// TIA Portal V16 export
// export: Created 2020-03-18T17:51:55.5456973Z, ExportSetting None, DisplayName Totally Integrated Automation Portal, DisplayVersion V16, DisplayName TIA Portal Version Control Interface, DisplayVersion V16, DisplayName TIA Portal Openness, DisplayVersion V16, DisplayName STEP 7 Professional, DisplayVersion V16, DisplayName STEP 7 Safety, DisplayVersion V16, DisplayName WinCC Advanced, DisplayVersion V16
DATA_BLOCK "DB_R134a_1_StepData"   // DB1310
{ S7_Optimized_Access := 'TRUE' }
AUTHOR : JMP/CSS
VERSION : 7.1
// stored: AutoNumber false, MemoryReserve 100
   VAR RETAIN
      Timestamp : Date_And_Time := DT#2019-07-18-09:28:16;
      DescriptionMedium : Array[1..4] of WString[36];
      "Step" { S7_SetPoint := 'True'} : Array[0..68] of "UDT_STEP_DATA";
      Values { S7_SetPoint := 'True'} : "UDT_CYCLE_VALUES";
      Valve { S7_SetPoint := 'True'} : Array[1..64] of "UDT_VISU_VALVE_NAMES";
      ParaInfo { S7_SetPoint := 'True'} : Array[1..15] of "UDT_STEP_DATA_PARA_VISU";
   END_VAR
BEGIN
   DescriptionMedium[1..2] := WSTRING#'R134a';
   DescriptionMedium[3] := WSTRING#'空调r134a';
   DescriptionMedium[4] := WSTRING#'Übersetzung fehlt';
   "Step"[0].NextStep := 4;
   "Step"[1..3].NextStep := 0;
   "Step"[4].NextStep := 10;
   "Step"[5..9].NextStep := 0;
   "Step"[10].NextStep := 11;
   "Step"[11].NextStep := 15;
   "Step"[12..14].NextStep := 0;
   "Step"[15].NextStep := 16;
   "Step"[16].NextStep := 20;
   "Step"[17].NextStep := 62;
   "Step"[18..19].NextStep := 0;
   "Step"[20].NextStep := 21;
   "Step"[21].NextStep := 22;
   "Step"[22].NextStep := 27;
   "Step"[23..26].NextStep := 0;
   "Step"[27].NextStep := 28;
   "Step"[28].NextStep := 29;
   "Step"[29].NextStep := 30;
   "Step"[30].NextStep := 31;
   "Step"[31].NextStep := 32;
   "Step"[32].NextStep := 33;
   "Step"[33].NextStep := 34;
   "Step"[34].NextStep := 35;
   "Step"[35].NextStep := 36;
   "Step"[36].NextStep := 37;
   "Step"[37].NextStep := 38;
   "Step"[38].NextStep := 39;
   "Step"[39].NextStep := 62;
   "Step"[40..61].NextStep := 0;
   "Step"[62].NextStep := 64;
   "Step"[63].NextStep := 0;
   "Step"[64].NextStep := 66;
   "Step"[65..68].NextStep := 0;
   "Step"[0..9].AbortStep := 0;
   "Step"[10..11].AbortStep := 62;
   "Step"[12..14].AbortStep := 0;
   "Step"[15].AbortStep := 62;
   "Step"[16].AbortStep := 17;
   "Step"[17].AbortStep := 62;
   "Step"[18..19].AbortStep := 0;
   "Step"[20..22].AbortStep := 27;
   "Step"[23..26].AbortStep := 0;
   "Step"[27].AbortStep := 28;
   "Step"[28..29].AbortStep := 62;
   "Step"[30..37].AbortStep := 17;
   "Step"[38].AbortStep := 39;
   "Step"[39].AbortStep := 62;
   "Step"[40..61].AbortStep := 0;
   "Step"[62].AbortStep := 64;
   "Step"[63..68].AbortStep := 0;
   "Step"[0..9].OptionStep := 0;
   "Step"[10].OptionStep := 15;
   "Step"[11..15].OptionStep := 0;
   "Step"[16].OptionStep := 29;
   "Step"[17..34].OptionStep := 0;
   "Step"[35].OptionStep := 37;
   "Step"[36].OptionStep := 0;
   "Step"[37].OptionStep := 57;
   "Step"[38..68].OptionStep := 0;
   "Step"[0..9].WaitingTime := 0;
   "Step"[10..11].WaitingTime := 1000;
   "Step"[12..14].WaitingTime := 0;
   "Step"[15].WaitingTime := 1000;
   "Step"[16].WaitingTime := 3000;
   "Step"[17].WaitingTime := 5000;
   "Step"[18..19].WaitingTime := 0;
   "Step"[20].WaitingTime := 20000;
   "Step"[21].WaitingTime := 10000;
   "Step"[22].WaitingTime := 5000;
   "Step"[23..26].WaitingTime := 0;
   "Step"[27..28].WaitingTime := 5000;
   "Step"[29].WaitingTime := 4000;
   "Step"[30].WaitingTime := 10000;
   "Step"[31].WaitingTime := 15000;
   "Step"[32].WaitingTime := 1000;
   "Step"[33].WaitingTime := 4000;
   "Step"[34].WaitingTime := 5000;
   "Step"[35..36].WaitingTime := 1000;
   "Step"[37].WaitingTime := 0;
   "Step"[38].WaitingTime := 1000;
   "Step"[39].WaitingTime := 2000;
   "Step"[40..65].WaitingTime := 0;
   "Step"[66].WaitingTime := 5000;
   "Step"[67..68].WaitingTime := 0;
   "Step"[0..10].MonitoringTime := 0;
   "Step"[11].MonitoringTime := 4000;
   "Step"[12..15].MonitoringTime := 0;
   "Step"[16].MonitoringTime := 4000;
   "Step"[17..19].MonitoringTime := 0;
   "Step"[20].MonitoringTime := 23000;
   "Step"[21].MonitoringTime := 11000;
   "Step"[22].MonitoringTime := 6000;
   "Step"[23..26].MonitoringTime := 0;
   "Step"[27..28].MonitoringTime := 10000;
   "Step"[29].MonitoringTime := 5000;
   "Step"[30].MonitoringTime := 15000;
   "Step"[31].MonitoringTime := 45000;
   "Step"[32].MonitoringTime := 0;
   "Step"[33..34].MonitoringTime := 6000;
   "Step"[35].MonitoringTime := 0;
   "Step"[36].MonitoringTime := 20000;
   "Step"[37].MonitoringTime := 0;
   "Step"[38].MonitoringTime := 20000;
   "Step"[39..68].MonitoringTime := 0;
   "Step"[0].Setpoint[0..15] := 0;
   "Step"[1].Setpoint[0..15] := 0;
   "Step"[2].Setpoint[0..15] := 0;
   "Step"[3].Setpoint[0..15] := 0;
   "Step"[4].Setpoint[0..15] := 0;
   "Step"[5].Setpoint[0..15] := 0;
   "Step"[6].Setpoint[0..15] := 0;
   "Step"[7].Setpoint[0..15] := 0;
   "Step"[8].Setpoint[0..15] := 0;
   "Step"[9].Setpoint[0..15] := 0;
   "Step"[10].Setpoint[0..15] := 0;
   "Step"[11].Setpoint[0] := 0;
   "Step"[11].Setpoint[1] := 100;
   "Step"[11].Setpoint[2..15] := 0;
   "Step"[12].Setpoint[0..15] := 0;
   "Step"[13].Setpoint[0..15] := 0;
   "Step"[14].Setpoint[0..15] := 0;
   "Step"[15].Setpoint[0..15] := 0;
   "Step"[16].Setpoint[0..4] := 0;
   "Step"[16].Setpoint[5] := 1200;
   "Step"[16].Setpoint[6..15] := 0;
   "Step"[17].Setpoint[0..15] := 0;
   "Step"[18].Setpoint[0..15] := 0;
   "Step"[19].Setpoint[0..15] := 0;
   "Step"[20].Setpoint[0..4] := 0;
   "Step"[20].Setpoint[5] := 15000;
   "Step"[20].Setpoint[6..12] := 0;
   "Step"[20].Setpoint[13] := 15200;
   "Step"[20].Setpoint[14..15] := 0;
   "Step"[21].Setpoint[0..4] := 0;
   "Step"[21].Setpoint[5] := 15000;
   "Step"[21].Setpoint[6..12] := 0;
   "Step"[21].Setpoint[13] := 15200;
   "Step"[21].Setpoint[14..15] := 0;
   "Step"[22].Setpoint[0..4] := 0;
   "Step"[22].Setpoint[5] := 14900;
   "Step"[22].Setpoint[6] := -100;
   "Step"[22].Setpoint[7..12] := 0;
   "Step"[22].Setpoint[13] := 15200;
   "Step"[22].Setpoint[14..15] := 0;
   "Step"[23].Setpoint[0..15] := 0;
   "Step"[24].Setpoint[0..15] := 0;
   "Step"[25].Setpoint[0..15] := 0;
   "Step"[26].Setpoint[0..15] := 0;
   "Step"[27].Setpoint[0..4] := 0;
   "Step"[27].Setpoint[5] := 3000;
   "Step"[27].Setpoint[6..15] := 0;
   "Step"[28].Setpoint[0..4] := 0;
   "Step"[28].Setpoint[5] := 500;
   "Step"[28].Setpoint[6..15] := 0;
   "Step"[29].Setpoint[0] := 0;
   "Step"[29].Setpoint[1] := 10;
   "Step"[29].Setpoint[2..15] := 0;
   "Step"[30].Setpoint[0] := 0;
   "Step"[30].Setpoint[1] := 500;
   "Step"[30].Setpoint[2..15] := 0;
   "Step"[31].Setpoint[0] := 0;
   "Step"[31].Setpoint[1] := 30;
   "Step"[31].Setpoint[2..15] := 0;
   "Step"[32].Setpoint[0..15] := 0;
   "Step"[33].Setpoint[0] := 0;
   "Step"[33].Setpoint[1] := 50;
   "Step"[33].Setpoint[2] := 40;
   "Step"[33].Setpoint[3..15] := 0;
   "Step"[34].Setpoint[0] := 0;
   "Step"[34].Setpoint[1] := 50;
   "Step"[34].Setpoint[2..15] := 0;
   "Step"[35].Setpoint[0..15] := 0;
   "Step"[36].Setpoint[0..7] := 0;
   "Step"[36].Setpoint[8] := 15;
   "Step"[36].Setpoint[9..15] := 0;
   "Step"[37].Setpoint[0..15] := 0;
   "Step"[38].Setpoint[0..6] := 0;
   "Step"[38].Setpoint[7] := 550;
   "Step"[38].Setpoint[8..15] := 0;
   "Step"[39].Setpoint[0..15] := 0;
   "Step"[40].Setpoint[0..15] := 0;
   "Step"[41].Setpoint[0..15] := 0;
   "Step"[42].Setpoint[0..15] := 0;
   "Step"[43].Setpoint[0..15] := 0;
   "Step"[44].Setpoint[0..15] := 0;
   "Step"[45].Setpoint[0..15] := 0;
   "Step"[46].Setpoint[0..15] := 0;
   "Step"[47].Setpoint[0..15] := 0;
   "Step"[48].Setpoint[0..15] := 0;
   "Step"[49].Setpoint[0..15] := 0;
   "Step"[50].Setpoint[0..15] := 0;
   "Step"[51].Setpoint[0..15] := 0;
   "Step"[52].Setpoint[0..15] := 0;
   "Step"[53].Setpoint[0..15] := 0;
   "Step"[54].Setpoint[0..15] := 0;
   "Step"[55].Setpoint[0..15] := 0;
   "Step"[56].Setpoint[0..15] := 0;
   "Step"[57].Setpoint[0..15] := 0;
   "Step"[58].Setpoint[0..15] := 0;
   "Step"[59].Setpoint[0..15] := 0;
   "Step"[60].Setpoint[0..15] := 0;
   "Step"[61].Setpoint[0..15] := 0;
   "Step"[62].Setpoint[0..15] := 0;
   "Step"[63].Setpoint[0..15] := 0;
   "Step"[64].Setpoint[0..15] := 0;
   "Step"[65].Setpoint[0..15] := 0;
   "Step"[66].Setpoint[0..15] := 0;
   "Step"[67].Setpoint[0..15] := 0;
   "Step"[68].Setpoint[0..15] := 0;
   "Step"[0..9].History.ElapsedTime := 0;
   "Step"[10..11].History.ElapsedTime := 1001;
   "Step"[12..14].History.ElapsedTime := 0;
   "Step"[15].History.ElapsedTime := 1001;
   "Step"[16].History.ElapsedTime := 3001;
   "Step"[17..19].History.ElapsedTime := 0;
   "Step"[20].History.ElapsedTime := 20001;
   "Step"[21].History.ElapsedTime := 10001;
   "Step"[22].History.ElapsedTime := 5001;
   "Step"[23..26].History.ElapsedTime := 0;
   "Step"[27..28].History.ElapsedTime := 5001;
   "Step"[29].History.ElapsedTime := 4001;
   "Step"[30].History.ElapsedTime := 10001;
   "Step"[31].History.ElapsedTime := 15001;
   "Step"[32].History.ElapsedTime := 1001;
   "Step"[33].History.ElapsedTime := 4001;
   "Step"[34].History.ElapsedTime := 5001;
   "Step"[35].History.ElapsedTime := 1001;
   "Step"[36].History.ElapsedTime := 3545;
   "Step"[37].History.ElapsedTime := 1;
   "Step"[38..61].History.ElapsedTime := 0;
   "Step"[62].History.ElapsedTime := 65252;
   "Step"[63].History.ElapsedTime := 0;
   "Step"[64].History.ElapsedTime := 7412;
   "Step"[65].History.ElapsedTime := 0;
   "Step"[66].History.ElapsedTime := 5001;
   "Step"[67..68].History.ElapsedTime := 0;
   "Step"[0].History.Values[0] := 0;
   "Step"[0].History.Values[1] := 6;
   "Step"[0].History.Values[2] := 0;
   "Step"[0].History.Values[3] := 15522;
   "Step"[0].History.Values[4] := -1;
   "Step"[0].History.Values[5] := 54;
   "Step"[0].History.Values[6] := -1;
   "Step"[0].History.Values[7] := 0;
   "Step"[0].History.Values[8] := 15;
   "Step"[0].History.Values[9..15] := 0;
   "Step"[1].History.Values[0..15] := 0;
   "Step"[2].History.Values[0..15] := 0;
   "Step"[3].History.Values[0..15] := 0;
   "Step"[4].History.Values[0..15] := 0;
   "Step"[5].History.Values[0..15] := 0;
   "Step"[6].History.Values[0..15] := 0;
   "Step"[7].History.Values[0..15] := 0;
   "Step"[8].History.Values[0..15] := 0;
   "Step"[9].History.Values[0..15] := 0;
   "Step"[10].History.Values[0] := 0;
   "Step"[10].History.Values[1..2] := 7;
   "Step"[10].History.Values[3..4] := 15524;
   "Step"[10].History.Values[5..6] := -700;
   "Step"[10].History.Values[7..15] := 0;
   "Step"[11].History.Values[0] := 0;
   "Step"[11].History.Values[1] := 10;
   "Step"[11].History.Values[2] := 3;
   "Step"[11].History.Values[3] := 15524;
   "Step"[11].History.Values[4] := 0;
   "Step"[11].History.Values[5] := -700;
   "Step"[11].History.Values[6..15] := 0;
   "Step"[12].History.Values[0..15] := 0;
   "Step"[13].History.Values[0..15] := 0;
   "Step"[14].History.Values[0..15] := 0;
   "Step"[15].History.Values[0] := 0;
   "Step"[15].History.Values[1] := 7;
   "Step"[15].History.Values[2] := -3;
   "Step"[15].History.Values[3] := 15524;
   "Step"[15].History.Values[4] := 0;
   "Step"[15].History.Values[5] := -700;
   "Step"[15].History.Values[6..15] := 0;
   "Step"[16].History.Values[0] := 0;
   "Step"[16].History.Values[1] := 6;
   "Step"[16].History.Values[2] := -1;
   "Step"[16].History.Values[3] := 15524;
   "Step"[16].History.Values[4] := 0;
   "Step"[16].History.Values[5] := -40;
   "Step"[16].History.Values[6] := 660;
   "Step"[16].History.Values[7..15] := 0;
   "Step"[17].History.Values[0..15] := 0;
   "Step"[18].History.Values[0..15] := 0;
   "Step"[19].History.Values[0..15] := 0;
   "Step"[20].History.Values[0] := 0;
   "Step"[20].History.Values[1] := 6;
   "Step"[20].History.Values[2] := 0;
   "Step"[20].History.Values[3] := 15524;
   "Step"[20].History.Values[4] := 0;
   "Step"[20].History.Values[5] := 15231;
   "Step"[20].History.Values[6] := 15271;
   "Step"[20].History.Values[7..12] := 0;
   "Step"[20].History.Values[13] := 15200;
   "Step"[20].History.Values[14..15] := 0;
   "Step"[21].History.Values[0] := 0;
   "Step"[21].History.Values[1] := 6;
   "Step"[21].History.Values[2] := 0;
   "Step"[21].History.Values[3] := 15523;
   "Step"[21].History.Values[4] := -1;
   "Step"[21].History.Values[5] := 15230;
   "Step"[21].History.Values[6] := -1;
   "Step"[21].History.Values[7..12] := 0;
   "Step"[21].History.Values[13] := 15200;
   "Step"[21].History.Values[14..15] := 0;
   "Step"[22].History.Values[0] := 0;
   "Step"[22].History.Values[1] := 6;
   "Step"[22].History.Values[2] := 0;
   "Step"[22].History.Values[3] := 15524;
   "Step"[22].History.Values[4] := 1;
   "Step"[22].History.Values[5] := 15231;
   "Step"[22].History.Values[6] := 1;
   "Step"[22].History.Values[7..12] := 0;
   "Step"[22].History.Values[13] := 15200;
   "Step"[22].History.Values[14..15] := 0;
   "Step"[23].History.Values[0..15] := 0;
   "Step"[24].History.Values[0..15] := 0;
   "Step"[25].History.Values[0..15] := 0;
   "Step"[26].History.Values[0..15] := 0;
   "Step"[27].History.Values[0] := 0;
   "Step"[27].History.Values[1] := 6;
   "Step"[27].History.Values[2] := 0;
   "Step"[27].History.Values[3] := 15523;
   "Step"[27].History.Values[4] := -1;
   "Step"[27].History.Values[5] := 46;
   "Step"[27].History.Values[6] := -15185;
   "Step"[27].History.Values[7..15] := 0;
   "Step"[28].History.Values[0] := 0;
   "Step"[28].History.Values[1] := 6;
   "Step"[28].History.Values[2] := 0;
   "Step"[28].History.Values[3] := 15523;
   "Step"[28].History.Values[4] := 0;
   "Step"[28].History.Values[5] := 47;
   "Step"[28].History.Values[6] := 1;
   "Step"[28].History.Values[7..15] := 0;
   "Step"[29].History.Values[0] := 0;
   "Step"[29].History.Values[1] := 19;
   "Step"[29].History.Values[2] := 13;
   "Step"[29].History.Values[3] := 15523;
   "Step"[29].History.Values[4] := 0;
   "Step"[29].History.Values[5] := -722;
   "Step"[29].History.Values[6] := -769;
   "Step"[29].History.Values[7..15] := 0;
   "Step"[30].History.Values[0] := 0;
   "Step"[30].History.Values[1] := 13;
   "Step"[30].History.Values[2] := -6;
   "Step"[30].History.Values[3] := 15523;
   "Step"[30].History.Values[4] := 0;
   "Step"[30].History.Values[5] := -716;
   "Step"[30].History.Values[6] := 6;
   "Step"[30].History.Values[7..15] := 0;
   "Step"[31].History.Values[0] := 0;
   "Step"[31].History.Values[1] := 10;
   "Step"[31].History.Values[2] := -3;
   "Step"[31].History.Values[3] := 15523;
   "Step"[31].History.Values[4] := 0;
   "Step"[31].History.Values[5] := -712;
   "Step"[31].History.Values[6] := 4;
   "Step"[31].History.Values[7..15] := 0;
   "Step"[32].History.Values[0] := 0;
   "Step"[32].History.Values[1] := 14;
   "Step"[32].History.Values[2] := 4;
   "Step"[32].History.Values[3] := 15523;
   "Step"[32].History.Values[4] := 0;
   "Step"[32].History.Values[5] := -711;
   "Step"[32].History.Values[6] := 1;
   "Step"[32].History.Values[7..15] := 0;
   "Step"[33].History.Values[0] := 0;
   "Step"[33].History.Values[1] := 22;
   "Step"[33].History.Values[2] := 8;
   "Step"[33].History.Values[3] := 15523;
   "Step"[33].History.Values[4] := 0;
   "Step"[33].History.Values[5] := -710;
   "Step"[33].History.Values[6] := 1;
   "Step"[33].History.Values[7..15] := 0;
   "Step"[34].History.Values[0] := 0;
   "Step"[34].History.Values[1] := 10;
   "Step"[34].History.Values[2] := -12;
   "Step"[34].History.Values[3] := 15523;
   "Step"[34].History.Values[4] := 0;
   "Step"[34].History.Values[5] := -710;
   "Step"[34].History.Values[6..15] := 0;
   "Step"[35].History.Values[0] := 0;
   "Step"[35].History.Values[1] := 7;
   "Step"[35].History.Values[2] := -3;
   "Step"[35].History.Values[3] := 15523;
   "Step"[35].History.Values[4] := 0;
   "Step"[35].History.Values[5] := -709;
   "Step"[35].History.Values[6] := 1;
   "Step"[35].History.Values[7..15] := 0;
   "Step"[36].History.Values[0] := 0;
   "Step"[36].History.Values[1] := 6;
   "Step"[36].History.Values[2] := -1;
   "Step"[36].History.Values[3] := 15523;
   "Step"[36].History.Values[4] := 0;
   "Step"[36].History.Values[5] := -708;
   "Step"[36].History.Values[6] := 1;
   "Step"[36].History.Values[7] := 0;
   "Step"[36].History.Values[8] := 14;
   "Step"[36].History.Values[9..15] := 0;
   "Step"[37].History.Values[0] := 0;
   "Step"[37].History.Values[1] := 6;
   "Step"[37].History.Values[2] := 0;
   "Step"[37].History.Values[3] := 15523;
   "Step"[37].History.Values[4] := 0;
   "Step"[37].History.Values[5] := -708;
   "Step"[37].History.Values[6..7] := 0;
   "Step"[37].History.Values[8] := 15;
   "Step"[37].History.Values[9..15] := 0;
   "Step"[38].History.Values[0..15] := 0;
   "Step"[39].History.Values[0..15] := 0;
   "Step"[40].History.Values[0..15] := 0;
   "Step"[41].History.Values[0..15] := 0;
   "Step"[42].History.Values[0..15] := 0;
   "Step"[43].History.Values[0..15] := 0;
   "Step"[44].History.Values[0..15] := 0;
   "Step"[45].History.Values[0..15] := 0;
   "Step"[46].History.Values[0..15] := 0;
   "Step"[47].History.Values[0..15] := 0;
   "Step"[48].History.Values[0..15] := 0;
   "Step"[49].History.Values[0..15] := 0;
   "Step"[50].History.Values[0..15] := 0;
   "Step"[51].History.Values[0..15] := 0;
   "Step"[52].History.Values[0..15] := 0;
   "Step"[53].History.Values[0..15] := 0;
   "Step"[54].History.Values[0..15] := 0;
   "Step"[55].History.Values[0..15] := 0;
   "Step"[56].History.Values[0..15] := 0;
   "Step"[57].History.Values[0..15] := 0;
   "Step"[58].History.Values[0..15] := 0;
   "Step"[59].History.Values[0..15] := 0;
   "Step"[60].History.Values[0..15] := 0;
   "Step"[61].History.Values[0..15] := 0;
   "Step"[62].History.Values[0] := 0;
   "Step"[62].History.Values[1] := 6;
   "Step"[62].History.Values[2] := 0;
   "Step"[62].History.Values[3] := 15523;
   "Step"[62].History.Values[4] := 0;
   "Step"[62].History.Values[5] := -698;
   "Step"[62].History.Values[6] := 10;
   "Step"[62].History.Values[7] := 0;
   "Step"[62].History.Values[8] := 15;
   "Step"[62].History.Values[9..15] := 0;
   "Step"[63].History.Values[0..15] := 0;
   "Step"[64].History.Values[0] := 0;
   "Step"[64].History.Values[1] := 6;
   "Step"[64].History.Values[2] := 0;
   "Step"[64].History.Values[3] := 15523;
   "Step"[64].History.Values[4] := 0;
   "Step"[64].History.Values[5] := 55;
   "Step"[64].History.Values[6] := 753;
   "Step"[64].History.Values[7] := 0;
   "Step"[64].History.Values[8] := 15;
   "Step"[64].History.Values[9..15] := 0;
   "Step"[65].History.Values[0..15] := 0;
   "Step"[66].History.Values[0] := 0;
   "Step"[66].History.Values[1] := 6;
   "Step"[66].History.Values[2] := 0;
   "Step"[66].History.Values[3] := 15522;
   "Step"[66].History.Values[4] := -1;
   "Step"[66].History.Values[5] := 54;
   "Step"[66].History.Values[6] := -1;
   "Step"[66].History.Values[7] := 0;
   "Step"[66].History.Values[8] := 15;
   "Step"[66].History.Values[9..15] := 0;
   "Step"[67].History.Values[0..15] := 0;
   "Step"[68].History.Values[0..15] := 0;
   "Step"[0].Valve[0..9] := FALSE;
   "Step"[0].Valve[10] := TRUE;
   "Step"[0].Valve[11] := FALSE;
   "Step"[0].Valve[12] := TRUE;
   "Step"[0].Valve[13..15] := FALSE;
   "Step"[0].Valve[16..21] := TRUE;
   "Step"[0].Valve[22] := FALSE;
   "Step"[0].Valve[23..24] := TRUE;
   "Step"[0].Valve[25..42] := FALSE;
   "Step"[0].Valve[43..45] := TRUE;
   "Step"[0].Valve[46..64] := FALSE;
   "Step"[1].Valve[0..64] := FALSE;
   "Step"[2].Valve[0..64] := FALSE;
   "Step"[3].Valve[0..64] := FALSE;
   "Step"[4].Valve[0..9] := FALSE;
   "Step"[4].Valve[10] := TRUE;
   "Step"[4].Valve[11] := FALSE;
   "Step"[4].Valve[12] := TRUE;
   "Step"[4].Valve[13..15] := FALSE;
   "Step"[4].Valve[16..21] := TRUE;
   "Step"[4].Valve[22] := FALSE;
   "Step"[4].Valve[23..24] := TRUE;
   "Step"[4].Valve[25..42] := FALSE;
   "Step"[4].Valve[43..46] := TRUE;
   "Step"[4].Valve[47..52] := FALSE;
   "Step"[4].Valve[53] := TRUE;
   "Step"[4].Valve[54..59] := FALSE;
   "Step"[4].Valve[60] := TRUE;
   "Step"[4].Valve[61..64] := FALSE;
   "Step"[5].Valve[0..64] := FALSE;
   "Step"[6].Valve[0..64] := FALSE;
   "Step"[7].Valve[0..64] := FALSE;
   "Step"[8].Valve[0..64] := FALSE;
   "Step"[9].Valve[0..64] := FALSE;
   "Step"[10].Valve[0..9] := FALSE;
   "Step"[10].Valve[10] := TRUE;
   "Step"[10].Valve[11] := FALSE;
   "Step"[10].Valve[12] := TRUE;
   "Step"[10].Valve[13..15] := FALSE;
   "Step"[10].Valve[16..21] := TRUE;
   "Step"[10].Valve[22] := FALSE;
   "Step"[10].Valve[23..24] := TRUE;
   "Step"[10].Valve[25..42] := FALSE;
   "Step"[10].Valve[43..45] := TRUE;
   "Step"[10].Valve[46..56] := FALSE;
   "Step"[10].Valve[57] := TRUE;
   "Step"[10].Valve[58..61] := FALSE;
   "Step"[10].Valve[62] := TRUE;
   "Step"[10].Valve[63..64] := FALSE;
   "Step"[11].Valve[0..9] := FALSE;
   "Step"[11].Valve[10] := TRUE;
   "Step"[11].Valve[11] := FALSE;
   "Step"[11].Valve[12] := TRUE;
   "Step"[11].Valve[13..15] := FALSE;
   "Step"[11].Valve[16..21] := TRUE;
   "Step"[11].Valve[22] := FALSE;
   "Step"[11].Valve[23..24] := TRUE;
   "Step"[11].Valve[25..42] := FALSE;
   "Step"[11].Valve[43..46] := TRUE;
   "Step"[11].Valve[47..52] := FALSE;
   "Step"[11].Valve[53] := TRUE;
   "Step"[11].Valve[54..56] := FALSE;
   "Step"[11].Valve[57] := TRUE;
   "Step"[11].Valve[58..59] := FALSE;
   "Step"[11].Valve[60] := TRUE;
   "Step"[11].Valve[61] := FALSE;
   "Step"[11].Valve[62] := TRUE;
   "Step"[11].Valve[63..64] := FALSE;
   "Step"[12].Valve[0..64] := FALSE;
   "Step"[13].Valve[0..64] := FALSE;
   "Step"[14].Valve[0..64] := FALSE;
   "Step"[15].Valve[0..9] := FALSE;
   "Step"[15].Valve[10] := TRUE;
   "Step"[15].Valve[11] := FALSE;
   "Step"[15].Valve[12] := TRUE;
   "Step"[15].Valve[13..15] := FALSE;
   "Step"[15].Valve[16..21] := TRUE;
   "Step"[15].Valve[22] := FALSE;
   "Step"[15].Valve[23..24] := TRUE;
   "Step"[15].Valve[25..42] := FALSE;
   "Step"[15].Valve[43..45] := TRUE;
   "Step"[15].Valve[46..52] := FALSE;
   "Step"[15].Valve[53] := TRUE;
   "Step"[15].Valve[54..56] := FALSE;
   "Step"[15].Valve[57] := TRUE;
   "Step"[15].Valve[58..59] := FALSE;
   "Step"[15].Valve[60] := TRUE;
   "Step"[15].Valve[61] := FALSE;
   "Step"[15].Valve[62] := TRUE;
   "Step"[15].Valve[63..64] := FALSE;
   "Step"[16].Valve[0..9] := FALSE;
   "Step"[16].Valve[10] := TRUE;
   "Step"[16].Valve[11] := FALSE;
   "Step"[16].Valve[12] := TRUE;
   "Step"[16].Valve[13..15] := FALSE;
   "Step"[16].Valve[16..21] := TRUE;
   "Step"[16].Valve[22] := FALSE;
   "Step"[16].Valve[23..24] := TRUE;
   "Step"[16].Valve[25..42] := FALSE;
   "Step"[16].Valve[43..45] := TRUE;
   "Step"[16].Valve[46..52] := FALSE;
   "Step"[16].Valve[53] := TRUE;
   "Step"[16].Valve[54..55] := FALSE;
   "Step"[16].Valve[56..57] := TRUE;
   "Step"[16].Valve[58..59] := FALSE;
   "Step"[16].Valve[60..62] := TRUE;
   "Step"[16].Valve[63..64] := FALSE;
   "Step"[17].Valve[0..9] := FALSE;
   "Step"[17].Valve[10] := TRUE;
   "Step"[17].Valve[11] := FALSE;
   "Step"[17].Valve[12] := TRUE;
   "Step"[17].Valve[13..15] := FALSE;
   "Step"[17].Valve[16..21] := TRUE;
   "Step"[17].Valve[22] := FALSE;
   "Step"[17].Valve[23..24] := TRUE;
   "Step"[17].Valve[25..42] := FALSE;
   "Step"[17].Valve[43..45] := TRUE;
   "Step"[17].Valve[46..48] := FALSE;
   "Step"[17].Valve[49] := TRUE;
   "Step"[17].Valve[50..52] := FALSE;
   "Step"[17].Valve[53] := TRUE;
   "Step"[17].Valve[54..56] := FALSE;
   "Step"[17].Valve[57] := TRUE;
   "Step"[17].Valve[58..59] := FALSE;
   "Step"[17].Valve[60] := TRUE;
   "Step"[17].Valve[61] := FALSE;
   "Step"[17].Valve[62] := TRUE;
   "Step"[17].Valve[63..64] := FALSE;
   "Step"[18].Valve[0..64] := FALSE;
   "Step"[19].Valve[0..64] := FALSE;
   "Step"[20].Valve[0..9] := FALSE;
   "Step"[20].Valve[10] := TRUE;
   "Step"[20].Valve[11] := FALSE;
   "Step"[20].Valve[12] := TRUE;
   "Step"[20].Valve[13..15] := FALSE;
   "Step"[20].Valve[16..21] := TRUE;
   "Step"[20].Valve[22] := FALSE;
   "Step"[20].Valve[23..24] := TRUE;
   "Step"[20].Valve[25..42] := FALSE;
   "Step"[20].Valve[43..45] := TRUE;
   "Step"[20].Valve[46] := FALSE;
   "Step"[20].Valve[47] := TRUE;
   "Step"[20].Valve[48..52] := FALSE;
   "Step"[20].Valve[53] := TRUE;
   "Step"[20].Valve[54..55] := FALSE;
   "Step"[20].Valve[56..57] := TRUE;
   "Step"[20].Valve[58..59] := FALSE;
   "Step"[20].Valve[60..62] := TRUE;
   "Step"[20].Valve[63..64] := FALSE;
   "Step"[21].Valve[0..9] := FALSE;
   "Step"[21].Valve[10] := TRUE;
   "Step"[21].Valve[11] := FALSE;
   "Step"[21].Valve[12] := TRUE;
   "Step"[21].Valve[13..15] := FALSE;
   "Step"[21].Valve[16..21] := TRUE;
   "Step"[21].Valve[22] := FALSE;
   "Step"[21].Valve[23..24] := TRUE;
   "Step"[21].Valve[25..42] := FALSE;
   "Step"[21].Valve[43..45] := TRUE;
   "Step"[21].Valve[46] := FALSE;
   "Step"[21].Valve[47] := TRUE;
   "Step"[21].Valve[48..52] := FALSE;
   "Step"[21].Valve[53] := TRUE;
   "Step"[21].Valve[54..55] := FALSE;
   "Step"[21].Valve[56..57] := TRUE;
   "Step"[21].Valve[58..59] := FALSE;
   "Step"[21].Valve[60..62] := TRUE;
   "Step"[21].Valve[63..64] := FALSE;
   "Step"[22].Valve[0..9] := FALSE;
   "Step"[22].Valve[10] := TRUE;
   "Step"[22].Valve[11] := FALSE;
   "Step"[22].Valve[12] := TRUE;
   "Step"[22].Valve[13..15] := FALSE;
   "Step"[22].Valve[16..21] := TRUE;
   "Step"[22].Valve[22] := FALSE;
   "Step"[22].Valve[23..24] := TRUE;
   "Step"[22].Valve[25..42] := FALSE;
   "Step"[22].Valve[43..45] := TRUE;
   "Step"[22].Valve[46..52] := FALSE;
   "Step"[22].Valve[53] := TRUE;
   "Step"[22].Valve[54..55] := FALSE;
   "Step"[22].Valve[56..57] := TRUE;
   "Step"[22].Valve[58..59] := FALSE;
   "Step"[22].Valve[60..62] := TRUE;
   "Step"[22].Valve[63..64] := FALSE;
   "Step"[23].Valve[0..64] := FALSE;
   "Step"[24].Valve[0..64] := FALSE;
   "Step"[25].Valve[0..64] := FALSE;
   "Step"[26].Valve[0..64] := FALSE;
   "Step"[27].Valve[0..9] := FALSE;
   "Step"[27].Valve[10] := TRUE;
   "Step"[27].Valve[11] := FALSE;
   "Step"[27].Valve[12] := TRUE;
   "Step"[27].Valve[13..15] := FALSE;
   "Step"[27].Valve[16..21] := TRUE;
   "Step"[27].Valve[22] := FALSE;
   "Step"[27].Valve[23..24] := TRUE;
   "Step"[27].Valve[25..42] := FALSE;
   "Step"[27].Valve[43..45] := TRUE;
   "Step"[27].Valve[46..48] := FALSE;
   "Step"[27].Valve[49] := TRUE;
   "Step"[27].Valve[50..52] := FALSE;
   "Step"[27].Valve[53] := TRUE;
   "Step"[27].Valve[54..55] := FALSE;
   "Step"[27].Valve[56..57] := TRUE;
   "Step"[27].Valve[58..59] := FALSE;
   "Step"[27].Valve[60..62] := TRUE;
   "Step"[27].Valve[63..64] := FALSE;
   "Step"[28].Valve[0..9] := FALSE;
   "Step"[28].Valve[10] := TRUE;
   "Step"[28].Valve[11] := FALSE;
   "Step"[28].Valve[12] := TRUE;
   "Step"[28].Valve[13..15] := FALSE;
   "Step"[28].Valve[16..21] := TRUE;
   "Step"[28].Valve[22] := FALSE;
   "Step"[28].Valve[23..24] := TRUE;
   "Step"[28].Valve[25..42] := FALSE;
   "Step"[28].Valve[43..45] := TRUE;
   "Step"[28].Valve[46..48] := FALSE;
   "Step"[28].Valve[49] := TRUE;
   "Step"[28].Valve[50..52] := FALSE;
   "Step"[28].Valve[53] := TRUE;
   "Step"[28].Valve[54..55] := FALSE;
   "Step"[28].Valve[56..57] := TRUE;
   "Step"[28].Valve[58..59] := FALSE;
   "Step"[28].Valve[60..62] := TRUE;
   "Step"[28].Valve[63..64] := FALSE;
   "Step"[29].Valve[0..9] := FALSE;
   "Step"[29].Valve[10] := TRUE;
   "Step"[29].Valve[11] := FALSE;
   "Step"[29].Valve[12] := TRUE;
   "Step"[29].Valve[13..15] := FALSE;
   "Step"[29].Valve[16..21] := TRUE;
   "Step"[29].Valve[22] := FALSE;
   "Step"[29].Valve[23..24] := TRUE;
   "Step"[29].Valve[25..42] := FALSE;
   "Step"[29].Valve[43..46] := TRUE;
   "Step"[29].Valve[47..52] := FALSE;
   "Step"[29].Valve[53] := TRUE;
   "Step"[29].Valve[54..55] := FALSE;
   "Step"[29].Valve[56..57] := TRUE;
   "Step"[29].Valve[58..59] := FALSE;
   "Step"[29].Valve[60..62] := TRUE;
   "Step"[29].Valve[63..64] := FALSE;
   "Step"[30].Valve[0..9] := FALSE;
   "Step"[30].Valve[10] := TRUE;
   "Step"[30].Valve[11] := FALSE;
   "Step"[30].Valve[12] := TRUE;
   "Step"[30].Valve[13..15] := FALSE;
   "Step"[30].Valve[16..21] := TRUE;
   "Step"[30].Valve[22] := FALSE;
   "Step"[30].Valve[23..24] := TRUE;
   "Step"[30].Valve[25..42] := FALSE;
   "Step"[30].Valve[43..46] := TRUE;
   "Step"[30].Valve[47..52] := FALSE;
   "Step"[30].Valve[53] := TRUE;
   "Step"[30].Valve[54..55] := FALSE;
   "Step"[30].Valve[56..57] := TRUE;
   "Step"[30].Valve[58..59] := FALSE;
   "Step"[30].Valve[60..62] := TRUE;
   "Step"[30].Valve[63..64] := FALSE;
   "Step"[31].Valve[0..9] := FALSE;
   "Step"[31].Valve[10] := TRUE;
   "Step"[31].Valve[11] := FALSE;
   "Step"[31].Valve[12] := TRUE;
   "Step"[31].Valve[13..15] := FALSE;
   "Step"[31].Valve[16..21] := TRUE;
   "Step"[31].Valve[22] := FALSE;
   "Step"[31].Valve[23..24] := TRUE;
   "Step"[31].Valve[25..42] := FALSE;
   "Step"[31].Valve[43..46] := TRUE;
   "Step"[31].Valve[47..52] := FALSE;
   "Step"[31].Valve[53] := TRUE;
   "Step"[31].Valve[54..55] := FALSE;
   "Step"[31].Valve[56..57] := TRUE;
   "Step"[31].Valve[58..59] := FALSE;
   "Step"[31].Valve[60..62] := TRUE;
   "Step"[31].Valve[63..64] := FALSE;
   "Step"[32].Valve[0..9] := FALSE;
   "Step"[32].Valve[10] := TRUE;
   "Step"[32].Valve[11] := FALSE;
   "Step"[32].Valve[12] := TRUE;
   "Step"[32].Valve[13..15] := FALSE;
   "Step"[32].Valve[16..21] := TRUE;
   "Step"[32].Valve[22] := FALSE;
   "Step"[32].Valve[23..24] := TRUE;
   "Step"[32].Valve[25..42] := FALSE;
   "Step"[32].Valve[43..44] := TRUE;
   "Step"[32].Valve[45] := FALSE;
   "Step"[32].Valve[46] := TRUE;
   "Step"[32].Valve[47..52] := FALSE;
   "Step"[32].Valve[53] := TRUE;
   "Step"[32].Valve[54..55] := FALSE;
   "Step"[32].Valve[56..57] := TRUE;
   "Step"[32].Valve[58..59] := FALSE;
   "Step"[32].Valve[60..62] := TRUE;
   "Step"[32].Valve[63..64] := FALSE;
   "Step"[33].Valve[0..9] := FALSE;
   "Step"[33].Valve[10] := TRUE;
   "Step"[33].Valve[11] := FALSE;
   "Step"[33].Valve[12] := TRUE;
   "Step"[33].Valve[13..15] := FALSE;
   "Step"[33].Valve[16..21] := TRUE;
   "Step"[33].Valve[22..43] := FALSE;
   "Step"[33].Valve[44] := TRUE;
   "Step"[33].Valve[45] := FALSE;
   "Step"[33].Valve[46] := TRUE;
   "Step"[33].Valve[47..52] := FALSE;
   "Step"[33].Valve[53] := TRUE;
   "Step"[33].Valve[54..55] := FALSE;
   "Step"[33].Valve[56..57] := TRUE;
   "Step"[33].Valve[58..59] := FALSE;
   "Step"[33].Valve[60..62] := TRUE;
   "Step"[33].Valve[63..64] := FALSE;
   "Step"[34].Valve[0..9] := FALSE;
   "Step"[34].Valve[10] := TRUE;
   "Step"[34].Valve[11] := FALSE;
   "Step"[34].Valve[12] := TRUE;
   "Step"[34].Valve[13..15] := FALSE;
   "Step"[34].Valve[16..21] := TRUE;
   "Step"[34].Valve[22..30] := FALSE;
   "Step"[34].Valve[31] := TRUE;
   "Step"[34].Valve[32..43] := FALSE;
   "Step"[34].Valve[44..46] := TRUE;
   "Step"[34].Valve[47..52] := FALSE;
   "Step"[34].Valve[53] := TRUE;
   "Step"[34].Valve[54..55] := FALSE;
   "Step"[34].Valve[56..57] := TRUE;
   "Step"[34].Valve[58..59] := FALSE;
   "Step"[34].Valve[60..62] := TRUE;
   "Step"[34].Valve[63..64] := FALSE;
   "Step"[35].Valve[0..9] := FALSE;
   "Step"[35].Valve[10] := TRUE;
   "Step"[35].Valve[11] := FALSE;
   "Step"[35].Valve[12] := TRUE;
   "Step"[35].Valve[13..15] := FALSE;
   "Step"[35].Valve[16..21] := TRUE;
   "Step"[35].Valve[22..30] := FALSE;
   "Step"[35].Valve[31] := TRUE;
   "Step"[35].Valve[32..43] := FALSE;
   "Step"[35].Valve[44..45] := TRUE;
   "Step"[35].Valve[46..55] := FALSE;
   "Step"[35].Valve[56..57] := TRUE;
   "Step"[35].Valve[58..61] := FALSE;
   "Step"[35].Valve[62] := TRUE;
   "Step"[35].Valve[63..64] := FALSE;
   "Step"[36].Valve[0..9] := FALSE;
   "Step"[36].Valve[10] := TRUE;
   "Step"[36].Valve[11] := FALSE;
   "Step"[36].Valve[12] := TRUE;
   "Step"[36].Valve[13..15] := FALSE;
   "Step"[36].Valve[16..21] := TRUE;
   "Step"[36].Valve[22..30] := FALSE;
   "Step"[36].Valve[31] := TRUE;
   "Step"[36].Valve[32..43] := FALSE;
   "Step"[36].Valve[44..45] := TRUE;
   "Step"[36].Valve[46..54] := FALSE;
   "Step"[36].Valve[55..57] := TRUE;
   "Step"[36].Valve[58..61] := FALSE;
   "Step"[36].Valve[62] := TRUE;
   "Step"[36].Valve[63..64] := FALSE;
   "Step"[37].Valve[0..9] := FALSE;
   "Step"[37].Valve[10] := TRUE;
   "Step"[37].Valve[11] := FALSE;
   "Step"[37].Valve[12] := TRUE;
   "Step"[37].Valve[13..15] := FALSE;
   "Step"[37].Valve[16..21] := TRUE;
   "Step"[37].Valve[22..43] := FALSE;
   "Step"[37].Valve[44..45] := TRUE;
   "Step"[37].Valve[46..55] := FALSE;
   "Step"[37].Valve[56..57] := TRUE;
   "Step"[37].Valve[58..61] := FALSE;
   "Step"[37].Valve[62] := TRUE;
   "Step"[37].Valve[63..64] := FALSE;
   "Step"[38].Valve[0..9] := FALSE;
   "Step"[38].Valve[10] := TRUE;
   "Step"[38].Valve[11] := FALSE;
   "Step"[38].Valve[12] := TRUE;
   "Step"[38].Valve[13..15] := FALSE;
   "Step"[38].Valve[16..21] := TRUE;
   "Step"[38].Valve[22..43] := FALSE;
   "Step"[38].Valve[44..45] := TRUE;
   "Step"[38].Valve[46..53] := FALSE;
   "Step"[38].Valve[54] := TRUE;
   "Step"[38].Valve[55] := FALSE;
   "Step"[38].Valve[56..57] := TRUE;
   "Step"[38].Valve[58..61] := FALSE;
   "Step"[38].Valve[62] := TRUE;
   "Step"[38].Valve[63..64] := FALSE;
   "Step"[39].Valve[0..9] := FALSE;
   "Step"[39].Valve[10] := TRUE;
   "Step"[39].Valve[11] := FALSE;
   "Step"[39].Valve[12] := TRUE;
   "Step"[39].Valve[13..15] := FALSE;
   "Step"[39].Valve[16..21] := TRUE;
   "Step"[39].Valve[22..43] := FALSE;
   "Step"[39].Valve[44..45] := TRUE;
   "Step"[39].Valve[46..55] := FALSE;
   "Step"[39].Valve[56..57] := TRUE;
   "Step"[39].Valve[58..61] := FALSE;
   "Step"[39].Valve[62] := TRUE;
   "Step"[39].Valve[63..64] := FALSE;
   "Step"[40].Valve[0..64] := FALSE;
   "Step"[41].Valve[0..64] := FALSE;
   "Step"[42].Valve[0..64] := FALSE;
   "Step"[43].Valve[0..64] := FALSE;
   "Step"[44].Valve[0..64] := FALSE;
   "Step"[45].Valve[0..64] := FALSE;
   "Step"[46].Valve[0..64] := FALSE;
   "Step"[47].Valve[0..64] := FALSE;
   "Step"[48].Valve[0..64] := FALSE;
   "Step"[49].Valve[0..64] := FALSE;
   "Step"[50].Valve[0..64] := FALSE;
   "Step"[51].Valve[0..64] := FALSE;
   "Step"[52].Valve[0..64] := FALSE;
   "Step"[53].Valve[0..64] := FALSE;
   "Step"[54].Valve[0..64] := FALSE;
   "Step"[55].Valve[0..64] := FALSE;
   "Step"[56].Valve[0..64] := FALSE;
   "Step"[57].Valve[0..64] := FALSE;
   "Step"[58].Valve[0..64] := FALSE;
   "Step"[59].Valve[0..64] := FALSE;
   "Step"[60].Valve[0..64] := FALSE;
   "Step"[61].Valve[0..64] := FALSE;
   "Step"[62].Valve[0..9] := FALSE;
   "Step"[62].Valve[10] := TRUE;
   "Step"[62].Valve[11] := FALSE;
   "Step"[62].Valve[12] := TRUE;
   "Step"[62].Valve[13..15] := FALSE;
   "Step"[62].Valve[16..21] := TRUE;
   "Step"[62].Valve[22..44] := FALSE;
   "Step"[62].Valve[45] := TRUE;
   "Step"[62].Valve[46..56] := FALSE;
   "Step"[62].Valve[57] := TRUE;
   "Step"[62].Valve[58..61] := FALSE;
   "Step"[62].Valve[62] := TRUE;
   "Step"[62].Valve[63..64] := FALSE;
   "Step"[63].Valve[0..64] := FALSE;
   "Step"[64].Valve[0..9] := FALSE;
   "Step"[64].Valve[10] := TRUE;
   "Step"[64].Valve[11] := FALSE;
   "Step"[64].Valve[12] := TRUE;
   "Step"[64].Valve[13..15] := FALSE;
   "Step"[64].Valve[16..21] := TRUE;
   "Step"[64].Valve[22..44] := FALSE;
   "Step"[64].Valve[45] := TRUE;
   "Step"[64].Valve[46..52] := FALSE;
   "Step"[64].Valve[53] := TRUE;
   "Step"[64].Valve[54..59] := FALSE;
   "Step"[64].Valve[60] := TRUE;
   "Step"[64].Valve[61..64] := FALSE;
   "Step"[65].Valve[0..64] := FALSE;
   "Step"[66].Valve[0..9] := FALSE;
   "Step"[66].Valve[10] := TRUE;
   "Step"[66].Valve[11] := FALSE;
   "Step"[66].Valve[12] := TRUE;
   "Step"[66].Valve[13..15] := FALSE;
   "Step"[66].Valve[16..21] := TRUE;
   "Step"[66].Valve[22] := FALSE;
   "Step"[66].Valve[23..24] := TRUE;
   "Step"[66].Valve[25..42] := FALSE;
   "Step"[66].Valve[43..45] := TRUE;
   "Step"[66].Valve[46..52] := FALSE;
   "Step"[66].Valve[53] := TRUE;
   "Step"[66].Valve[54..59] := FALSE;
   "Step"[66].Valve[60] := TRUE;
   "Step"[66].Valve[61..64] := FALSE;
   "Step"[67].Valve[0..64] := FALSE;
   "Step"[68].Valve[0..64] := FALSE;
   "Step"[0].HMI.Stepname.Language[1] := WSTRING#'Standby';
   "Step"[0].HMI.Stepname.Language[2] := WSTRING#'stand by';
   "Step"[0].HMI.Stepname.Language[3..4] := WSTRING#'';
   "Step"[1].HMI.Stepname.Language[1..4] := WSTRING#'';
   "Step"[2].HMI.Stepname.Language[1..4] := WSTRING#'';
   "Step"[3].HMI.Stepname.Language[1..4] := WSTRING#'';
   "Step"[4].HMI.Stepname.Language[1] := WSTRING#'Adapter Belueften';
   "Step"[4].HMI.Stepname.Language[2] := WSTRING#'venting adapter';
   "Step"[4].HMI.Stepname.Language[3..4] := WSTRING#'';
   "Step"[5].HMI.Stepname.Language[1..4] := WSTRING#'';
   "Step"[6].HMI.Stepname.Language[1..4] := WSTRING#'';
   "Step"[7].HMI.Stepname.Language[1..4] := WSTRING#'';
   "Step"[8].HMI.Stepname.Language[1..4] := WSTRING#'';
   "Step"[9].HMI.Stepname.Language[1..4] := WSTRING#'';
   "Step"[10].HMI.Stepname.Language[1] := WSTRING#'Zyklus Start inkl. Verri';
   "Step"[10].HMI.Stepname.Language[2] := WSTRING#'cycle start';
   "Step"[10].HMI.Stepname.Language[3..4] := WSTRING#'';
   "Step"[11].HMI.Stepname.Language[1] := WSTRING#'Vakuumast evakuieren (Ad';
   "Step"[11].HMI.Stepname.Language[2] := WSTRING#'evacuating vacuumpipe';
   "Step"[11].HMI.Stepname.Language[3..4] := WSTRING#'';
   "Step"[12].HMI.Stepname.Language[1..4] := WSTRING#'';
   "Step"[13].HMI.Stepname.Language[1..4] := WSTRING#'';
   "Step"[14].HMI.Stepname.Language[1..4] := WSTRING#'';
   "Step"[15].HMI.Stepname.Language[1] := WSTRING#'Umschalten';
   "Step"[15].HMI.Stepname.Language[2] := WSTRING#'change sequence';
   "Step"[15].HMI.Stepname.Language[3..4] := WSTRING#'';
   "Step"[16].HMI.Stepname.Language[1] := WSTRING#'Systemtest 1 Druck';
   "Step"[16].HMI.Stepname.Language[2] := WSTRING#'systemtest 1 pressure';
   "Step"[16].HMI.Stepname.Language[3..4] := WSTRING#'';
   "Step"[17].HMI.Stepname.Language[1] := WSTRING#'System entlasten';
   "Step"[17].HMI.Stepname.Language[2] := WSTRING#'release system';
   "Step"[17].HMI.Stepname.Language[3..4] := WSTRING#'';
   "Step"[18].HMI.Stepname.Language[1..4] := WSTRING#'';
   "Step"[19].HMI.Stepname.Language[1..4] := WSTRING#'';
   "Step"[20].HMI.Stepname.Language[1] := WSTRING#'Druckluft Fuellen';
   "Step"[20].HMI.Stepname.Language[2] := WSTRING#'compr.air fill';
   "Step"[20].HMI.Stepname.Language[3..4] := WSTRING#'';
   "Step"[21].HMI.Stepname.Language[1] := WSTRING#'Druckluft Stabilisieren';
   "Step"[21].HMI.Stepname.Language[2] := WSTRING#'compr. air stabilize';
   "Step"[21].HMI.Stepname.Language[3..4] := WSTRING#'';
   "Step"[22].HMI.Stepname.Language[1] := WSTRING#'Drucklufttest';
   "Step"[22].HMI.Stepname.Language[2] := WSTRING#'compr. air test';
   "Step"[22].HMI.Stepname.Language[3..4] := WSTRING#'';
   "Step"[23].HMI.Stepname.Language[1..4] := WSTRING#'';
   "Step"[24].HMI.Stepname.Language[1..4] := WSTRING#'';
   "Step"[25].HMI.Stepname.Language[1..4] := WSTRING#'';
   "Step"[26].HMI.Stepname.Language[1..4] := WSTRING#'';
   "Step"[27].HMI.Stepname.Language[1] := WSTRING#'Druckluft entlasten 1';
   "Step"[27].HMI.Stepname.Language[2] := WSTRING#'compr. air release 1';
   "Step"[27].HMI.Stepname.Language[3..4] := WSTRING#'';
   "Step"[28].HMI.Stepname.Language[1] := WSTRING#'Druckluft entlasten 2';
   "Step"[28].HMI.Stepname.Language[2] := WSTRING#'compr. air release 2';
   "Step"[28].HMI.Stepname.Language[3..4] := WSTRING#'';
   "Step"[29].HMI.Stepname.Language[1] := WSTRING#'Test Schraderventil geoe';
   "Step"[29].HMI.Stepname.Language[2] := WSTRING#'test connection to vehic';
   "Step"[29].HMI.Stepname.Language[3..4] := WSTRING#'';
   "Step"[30].HMI.Stepname.Language[1] := WSTRING#'Evakuieren 1';
   "Step"[30].HMI.Stepname.Language[2] := WSTRING#'evacuation 1';
   "Step"[30].HMI.Stepname.Language[3..4] := WSTRING#'';
   "Step"[31].HMI.Stepname.Language[1] := WSTRING#'Evakuieren 2';
   "Step"[31].HMI.Stepname.Language[2] := WSTRING#'evacuation 2';
   "Step"[31].HMI.Stepname.Language[3..4] := WSTRING#'';
   "Step"[32].HMI.Stepname.Language[1] := WSTRING#'Evakuieren stabilisieren';
   "Step"[32].HMI.Stepname.Language[2] := WSTRING#'evacuation stabilize';
   "Step"[32].HMI.Stepname.Language[3..4] := WSTRING#'';
   "Step"[33].HMI.Stepname.Language[1] := WSTRING#'Vakuumtest';
   "Step"[33].HMI.Stepname.Language[2] := WSTRING#'vacuumtest';
   "Step"[33].HMI.Stepname.Language[3..4] := WSTRING#'';
   "Step"[34].HMI.Stepname.Language[1] := WSTRING#'Evakuieren 3';
   "Step"[34].HMI.Stepname.Language[2] := WSTRING#'evacuation 3';
   "Step"[34].HMI.Stepname.Language[3..4] := WSTRING#'';
   "Step"[35].HMI.Stepname.Language[1] := WSTRING#'Umschalten V/F';
   "Step"[35].HMI.Stepname.Language[2] := WSTRING#'change sequence V/F';
   "Step"[35].HMI.Stepname.Language[3..4] := WSTRING#'';
   "Step"[36].HMI.Stepname.Language[1] := WSTRING#'Fuellen 1 PAG-Oel (Volum';
   "Step"[36].HMI.Stepname.Language[2] := WSTRING#'filling 1 PAG oil';
   "Step"[36].HMI.Stepname.Language[3..4] := WSTRING#'';
   "Step"[37].HMI.Stepname.Language[1] := WSTRING#'Umschalten Fuellen PAG-O';
   "Step"[37].HMI.Stepname.Language[2] := WSTRING#'change sequence f1/f2';
   "Step"[37].HMI.Stepname.Language[3..4] := WSTRING#'';
   "Step"[38].HMI.Stepname.Language[1] := WSTRING#'Fuellen 2 R134a (Masse)';
   "Step"[38].HMI.Stepname.Language[2] := WSTRING#'filling 2 R134a';
   "Step"[38].HMI.Stepname.Language[3..4] := WSTRING#'';
   "Step"[39].HMI.Stepname.Language[1] := WSTRING#'Warten/Nachbereiten';
   "Step"[39].HMI.Stepname.Language[2] := WSTRING#'Waiting';
   "Step"[39].HMI.Stepname.Language[3..4] := WSTRING#'';
   "Step"[40].HMI.Stepname.Language[1..4] := WSTRING#'';
   "Step"[41].HMI.Stepname.Language[1..4] := WSTRING#'';
   "Step"[42].HMI.Stepname.Language[1..4] := WSTRING#'';
   "Step"[43].HMI.Stepname.Language[1..4] := WSTRING#'';
   "Step"[44].HMI.Stepname.Language[1..4] := WSTRING#'';
   "Step"[45].HMI.Stepname.Language[1..4] := WSTRING#'';
   "Step"[46].HMI.Stepname.Language[1..4] := WSTRING#'';
   "Step"[47].HMI.Stepname.Language[1..4] := WSTRING#'';
   "Step"[48].HMI.Stepname.Language[1..4] := WSTRING#'';
   "Step"[49].HMI.Stepname.Language[1..4] := WSTRING#'';
   "Step"[50].HMI.Stepname.Language[1..4] := WSTRING#'';
   "Step"[51].HMI.Stepname.Language[1..4] := WSTRING#'';
   "Step"[52].HMI.Stepname.Language[1..4] := WSTRING#'';
   "Step"[53].HMI.Stepname.Language[1..4] := WSTRING#'';
   "Step"[54].HMI.Stepname.Language[1..4] := WSTRING#'';
   "Step"[55].HMI.Stepname.Language[1..4] := WSTRING#'';
   "Step"[56].HMI.Stepname.Language[1..4] := WSTRING#'';
   "Step"[57].HMI.Stepname.Language[1..4] := WSTRING#'';
   "Step"[58].HMI.Stepname.Language[1..4] := WSTRING#'';
   "Step"[59].HMI.Stepname.Language[1..4] := WSTRING#'';
   "Step"[60].HMI.Stepname.Language[1..4] := WSTRING#'';
   "Step"[61].HMI.Stepname.Language[1..4] := WSTRING#'';
   "Step"[62].HMI.Stepname.Language[1] := WSTRING#'Zyklus Ende';
   "Step"[62].HMI.Stepname.Language[2] := WSTRING#'cycle end';
   "Step"[62].HMI.Stepname.Language[3..4] := WSTRING#'';
   "Step"[63].HMI.Stepname.Language[1..4] := WSTRING#'';
   "Step"[64].HMI.Stepname.Language[1] := WSTRING#'Warten 1';
   "Step"[64].HMI.Stepname.Language[2] := WSTRING#'wait for adapter home';
   "Step"[64].HMI.Stepname.Language[3..4] := WSTRING#'';
   "Step"[65].HMI.Stepname.Language[1..4] := WSTRING#'';
   "Step"[66].HMI.Stepname.Language[1] := WSTRING#'Schlaeuche reinigen';
   "Step"[66].HMI.Stepname.Language[2] := WSTRING#'clean hoses';
   "Step"[66].HMI.Stepname.Language[3..4] := WSTRING#'';
   "Step"[67].HMI.Stepname.Language[1..4] := WSTRING#'';
   "Step"[68].HMI.Stepname.Language[1..4] := WSTRING#'';
   "Step"[0].HMI.Stepname.Actual := WSTRING#'Standby';
   "Step"[1..3].HMI.Stepname.Actual := WSTRING#'';
   "Step"[4].HMI.Stepname.Actual := WSTRING#'Adapter Belueften';
   "Step"[5..9].HMI.Stepname.Actual := WSTRING#'';
   "Step"[10].HMI.Stepname.Actual := WSTRING#'Zyklus Start inkl. Verri';
   "Step"[11].HMI.Stepname.Actual := WSTRING#'Vakuumast evakuieren (Ad';
   "Step"[12..14].HMI.Stepname.Actual := WSTRING#'';
   "Step"[15].HMI.Stepname.Actual := WSTRING#'Umschalten';
   "Step"[16].HMI.Stepname.Actual := WSTRING#'Systemtest 1 Druck';
   "Step"[17].HMI.Stepname.Actual := WSTRING#'System entlasten';
   "Step"[18..19].HMI.Stepname.Actual := WSTRING#'';
   "Step"[20].HMI.Stepname.Actual := WSTRING#'Druckluft Fuellen';
   "Step"[21].HMI.Stepname.Actual := WSTRING#'Druckluft Stabilisieren';
   "Step"[22].HMI.Stepname.Actual := WSTRING#'Drucklufttest';
   "Step"[23..26].HMI.Stepname.Actual := WSTRING#'';
   "Step"[27].HMI.Stepname.Actual := WSTRING#'Druckluft entlasten 1';
   "Step"[28].HMI.Stepname.Actual := WSTRING#'Druckluft entlasten 2';
   "Step"[29].HMI.Stepname.Actual := WSTRING#'Test Schraderventil geoe';
   "Step"[30].HMI.Stepname.Actual := WSTRING#'Evakuieren 1';
   "Step"[31].HMI.Stepname.Actual := WSTRING#'Evakuieren 2';
   "Step"[32].HMI.Stepname.Actual := WSTRING#'Evakuieren stabilisieren';
   "Step"[33].HMI.Stepname.Actual := WSTRING#'Vakuumtest';
   "Step"[34].HMI.Stepname.Actual := WSTRING#'Evakuieren 3';
   "Step"[35].HMI.Stepname.Actual := WSTRING#'Umschalten V/F';
   "Step"[36].HMI.Stepname.Actual := WSTRING#'Fuellen 1 PAG-Oel (Volum';
   "Step"[37].HMI.Stepname.Actual := WSTRING#'Umschalten Fuellen PAG-O';
   "Step"[38].HMI.Stepname.Actual := WSTRING#'Fuellen 2 R134a (Masse)';
   "Step"[39].HMI.Stepname.Actual := WSTRING#'Warten/Nachbereiten';
   "Step"[40..61].HMI.Stepname.Actual := WSTRING#'';
   "Step"[62].HMI.Stepname.Actual := WSTRING#'Zyklus Ende';
   "Step"[63].HMI.Stepname.Actual := WSTRING#'';
   "Step"[64].HMI.Stepname.Actual := WSTRING#'Warten 1';
   "Step"[65].HMI.Stepname.Actual := WSTRING#'';
   "Step"[66].HMI.Stepname.Actual := WSTRING#'Schlaeuche reinigen';
   "Step"[67..68].HMI.Stepname.Actual := WSTRING#'';
   "Step"[0].HMI.Display.NextStep := TRUE;
   "Step"[1..3].HMI.Display.NextStep := FALSE;
   "Step"[4].HMI.Display.NextStep := TRUE;
   "Step"[5..9].HMI.Display.NextStep := FALSE;
   "Step"[10..11].HMI.Display.NextStep := TRUE;
   "Step"[12..14].HMI.Display.NextStep := FALSE;
   "Step"[15..17].HMI.Display.NextStep := TRUE;
   "Step"[18..19].HMI.Display.NextStep := FALSE;
   "Step"[20..22].HMI.Display.NextStep := TRUE;
   "Step"[23..26].HMI.Display.NextStep := FALSE;
   "Step"[27..39].HMI.Display.NextStep := TRUE;
   "Step"[40..61].HMI.Display.NextStep := FALSE;
   "Step"[62].HMI.Display.NextStep := TRUE;
   "Step"[63].HMI.Display.NextStep := FALSE;
   "Step"[64].HMI.Display.NextStep := TRUE;
   "Step"[65].HMI.Display.NextStep := FALSE;
   "Step"[66].HMI.Display.NextStep := TRUE;
   "Step"[67..68].HMI.Display.NextStep := FALSE;
   "Step"[0..9].HMI.Display.AbortStep := FALSE;
   "Step"[10..11].HMI.Display.AbortStep := TRUE;
   "Step"[12..14].HMI.Display.AbortStep := FALSE;
   "Step"[15..17].HMI.Display.AbortStep := TRUE;
   "Step"[18..19].HMI.Display.AbortStep := FALSE;
   "Step"[20..22].HMI.Display.AbortStep := TRUE;
   "Step"[23..26].HMI.Display.AbortStep := FALSE;
   "Step"[27..39].HMI.Display.AbortStep := TRUE;
   "Step"[40..61].HMI.Display.AbortStep := FALSE;
   "Step"[62].HMI.Display.AbortStep := TRUE;
   "Step"[63..68].HMI.Display.AbortStep := FALSE;
   "Step"[0..3].HMI.Display.OptionStep := FALSE;
   "Step"[4].HMI.Display.OptionStep := TRUE;
   "Step"[5..9].HMI.Display.OptionStep := FALSE;
   "Step"[10].HMI.Display.OptionStep := TRUE;
   "Step"[11..15].HMI.Display.OptionStep := FALSE;
   "Step"[16].HMI.Display.OptionStep := TRUE;
   "Step"[17..34].HMI.Display.OptionStep := FALSE;
   "Step"[35].HMI.Display.OptionStep := TRUE;
   "Step"[36].HMI.Display.OptionStep := FALSE;
   "Step"[37].HMI.Display.OptionStep := TRUE;
   "Step"[38..68].HMI.Display.OptionStep := FALSE;
   "Step"[0..9].HMI.Display.WaitingTime := FALSE;
   "Step"[10..11].HMI.Display.WaitingTime := TRUE;
   "Step"[12..14].HMI.Display.WaitingTime := FALSE;
   "Step"[15..17].HMI.Display.WaitingTime := TRUE;
   "Step"[18..19].HMI.Display.WaitingTime := FALSE;
   "Step"[20..22].HMI.Display.WaitingTime := TRUE;
   "Step"[23..26].HMI.Display.WaitingTime := FALSE;
   "Step"[27..39].HMI.Display.WaitingTime := TRUE;
   "Step"[40..65].HMI.Display.WaitingTime := FALSE;
   "Step"[66].HMI.Display.WaitingTime := TRUE;
   "Step"[67..68].HMI.Display.WaitingTime := FALSE;
   "Step"[0..10].HMI.Display.MonitoringTime := FALSE;
   "Step"[11].HMI.Display.MonitoringTime := TRUE;
   "Step"[12..15].HMI.Display.MonitoringTime := FALSE;
   "Step"[16].HMI.Display.MonitoringTime := TRUE;
   "Step"[17..19].HMI.Display.MonitoringTime := FALSE;
   "Step"[20..22].HMI.Display.MonitoringTime := TRUE;
   "Step"[23..26].HMI.Display.MonitoringTime := FALSE;
   "Step"[27..31].HMI.Display.MonitoringTime := TRUE;
   "Step"[32].HMI.Display.MonitoringTime := FALSE;
   "Step"[33].HMI.Display.MonitoringTime := TRUE;
   "Step"[34..35].HMI.Display.MonitoringTime := FALSE;
   "Step"[36].HMI.Display.MonitoringTime := TRUE;
   "Step"[37].HMI.Display.MonitoringTime := FALSE;
   "Step"[38].HMI.Display.MonitoringTime := TRUE;
   "Step"[39..68].HMI.Display.MonitoringTime := FALSE;
   "Step"[0].HMI.Display.Setpoint[0..12] := FALSE;
   "Step"[0].HMI.Display.Setpoint[13] := TRUE;
   "Step"[0].HMI.Display.Setpoint[14..15] := FALSE;
   "Step"[1].HMI.Display.Setpoint[0..15] := FALSE;
   "Step"[2].HMI.Display.Setpoint[0..15] := FALSE;
   "Step"[3].HMI.Display.Setpoint[0..15] := FALSE;
   "Step"[4].HMI.Display.Setpoint[0..12] := FALSE;
   "Step"[4].HMI.Display.Setpoint[13] := TRUE;
   "Step"[4].HMI.Display.Setpoint[14..15] := FALSE;
   "Step"[5].HMI.Display.Setpoint[0..15] := FALSE;
   "Step"[6].HMI.Display.Setpoint[0..15] := FALSE;
   "Step"[7].HMI.Display.Setpoint[0..15] := FALSE;
   "Step"[8].HMI.Display.Setpoint[0..15] := FALSE;
   "Step"[9].HMI.Display.Setpoint[0..15] := FALSE;
   "Step"[10].HMI.Display.Setpoint[0..12] := FALSE;
   "Step"[10].HMI.Display.Setpoint[13] := TRUE;
   "Step"[10].HMI.Display.Setpoint[14..15] := FALSE;
   "Step"[11].HMI.Display.Setpoint[0] := FALSE;
   "Step"[11].HMI.Display.Setpoint[1] := TRUE;
   "Step"[11].HMI.Display.Setpoint[2..12] := FALSE;
   "Step"[11].HMI.Display.Setpoint[13] := TRUE;
   "Step"[11].HMI.Display.Setpoint[14..15] := FALSE;
   "Step"[12].HMI.Display.Setpoint[0..15] := FALSE;
   "Step"[13].HMI.Display.Setpoint[0..15] := FALSE;
   "Step"[14].HMI.Display.Setpoint[0..15] := FALSE;
   "Step"[15].HMI.Display.Setpoint[0..12] := FALSE;
   "Step"[15].HMI.Display.Setpoint[13] := TRUE;
   "Step"[15].HMI.Display.Setpoint[14..15] := FALSE;
   "Step"[16].HMI.Display.Setpoint[0..4] := FALSE;
   "Step"[16].HMI.Display.Setpoint[5] := TRUE;
   "Step"[16].HMI.Display.Setpoint[6..12] := FALSE;
   "Step"[16].HMI.Display.Setpoint[13] := TRUE;
   "Step"[16].HMI.Display.Setpoint[14..15] := FALSE;
   "Step"[17].HMI.Display.Setpoint[0..12] := FALSE;
   "Step"[17].HMI.Display.Setpoint[13] := TRUE;
   "Step"[17].HMI.Display.Setpoint[14..15] := FALSE;
   "Step"[18].HMI.Display.Setpoint[0..15] := FALSE;
   "Step"[19].HMI.Display.Setpoint[0..15] := FALSE;
   "Step"[20].HMI.Display.Setpoint[0..4] := FALSE;
   "Step"[20].HMI.Display.Setpoint[5] := TRUE;
   "Step"[20].HMI.Display.Setpoint[6..12] := FALSE;
   "Step"[20].HMI.Display.Setpoint[13] := TRUE;
   "Step"[20].HMI.Display.Setpoint[14..15] := FALSE;
   "Step"[21].HMI.Display.Setpoint[0..4] := FALSE;
   "Step"[21].HMI.Display.Setpoint[5] := TRUE;
   "Step"[21].HMI.Display.Setpoint[6..12] := FALSE;
   "Step"[21].HMI.Display.Setpoint[13] := TRUE;
   "Step"[21].HMI.Display.Setpoint[14..15] := FALSE;
   "Step"[22].HMI.Display.Setpoint[0..4] := FALSE;
   "Step"[22].HMI.Display.Setpoint[5..6] := TRUE;
   "Step"[22].HMI.Display.Setpoint[7..12] := FALSE;
   "Step"[22].HMI.Display.Setpoint[13] := TRUE;
   "Step"[22].HMI.Display.Setpoint[14..15] := FALSE;
   "Step"[23].HMI.Display.Setpoint[0..15] := FALSE;
   "Step"[24].HMI.Display.Setpoint[0..15] := FALSE;
   "Step"[25].HMI.Display.Setpoint[0..15] := FALSE;
   "Step"[26].HMI.Display.Setpoint[0..15] := FALSE;
   "Step"[27].HMI.Display.Setpoint[0..4] := FALSE;
   "Step"[27].HMI.Display.Setpoint[5] := TRUE;
   "Step"[27].HMI.Display.Setpoint[6..12] := FALSE;
   "Step"[27].HMI.Display.Setpoint[13] := TRUE;
   "Step"[27].HMI.Display.Setpoint[14..15] := FALSE;
   "Step"[28].HMI.Display.Setpoint[0..4] := FALSE;
   "Step"[28].HMI.Display.Setpoint[5] := TRUE;
   "Step"[28].HMI.Display.Setpoint[6..12] := FALSE;
   "Step"[28].HMI.Display.Setpoint[13] := TRUE;
   "Step"[28].HMI.Display.Setpoint[14..15] := FALSE;
   "Step"[29].HMI.Display.Setpoint[0] := FALSE;
   "Step"[29].HMI.Display.Setpoint[1] := TRUE;
   "Step"[29].HMI.Display.Setpoint[2..12] := FALSE;
   "Step"[29].HMI.Display.Setpoint[13] := TRUE;
   "Step"[29].HMI.Display.Setpoint[14..15] := FALSE;
   "Step"[30].HMI.Display.Setpoint[0] := FALSE;
   "Step"[30].HMI.Display.Setpoint[1] := TRUE;
   "Step"[30].HMI.Display.Setpoint[2..12] := FALSE;
   "Step"[30].HMI.Display.Setpoint[13] := TRUE;
   "Step"[30].HMI.Display.Setpoint[14..15] := FALSE;
   "Step"[31].HMI.Display.Setpoint[0] := FALSE;
   "Step"[31].HMI.Display.Setpoint[1] := TRUE;
   "Step"[31].HMI.Display.Setpoint[2..12] := FALSE;
   "Step"[31].HMI.Display.Setpoint[13] := TRUE;
   "Step"[31].HMI.Display.Setpoint[14..15] := FALSE;
   "Step"[32].HMI.Display.Setpoint[0..12] := FALSE;
   "Step"[32].HMI.Display.Setpoint[13] := TRUE;
   "Step"[32].HMI.Display.Setpoint[14..15] := FALSE;
   "Step"[33].HMI.Display.Setpoint[0] := FALSE;
   "Step"[33].HMI.Display.Setpoint[1..2] := TRUE;
   "Step"[33].HMI.Display.Setpoint[3..12] := FALSE;
   "Step"[33].HMI.Display.Setpoint[13] := TRUE;
   "Step"[33].HMI.Display.Setpoint[14..15] := FALSE;
   "Step"[34].HMI.Display.Setpoint[0..12] := FALSE;
   "Step"[34].HMI.Display.Setpoint[13] := TRUE;
   "Step"[34].HMI.Display.Setpoint[14..15] := FALSE;
   "Step"[35].HMI.Display.Setpoint[0..12] := FALSE;
   "Step"[35].HMI.Display.Setpoint[13] := TRUE;
   "Step"[35].HMI.Display.Setpoint[14..15] := FALSE;
   "Step"[36].HMI.Display.Setpoint[0..7] := FALSE;
   "Step"[36].HMI.Display.Setpoint[8] := TRUE;
   "Step"[36].HMI.Display.Setpoint[9..12] := FALSE;
   "Step"[36].HMI.Display.Setpoint[13] := TRUE;
   "Step"[36].HMI.Display.Setpoint[14..15] := FALSE;
   "Step"[37].HMI.Display.Setpoint[0..12] := FALSE;
   "Step"[37].HMI.Display.Setpoint[13] := TRUE;
   "Step"[37].HMI.Display.Setpoint[14..15] := FALSE;
   "Step"[38].HMI.Display.Setpoint[0..6] := FALSE;
   "Step"[38].HMI.Display.Setpoint[7] := TRUE;
   "Step"[38].HMI.Display.Setpoint[8..12] := FALSE;
   "Step"[38].HMI.Display.Setpoint[13] := TRUE;
   "Step"[38].HMI.Display.Setpoint[14..15] := FALSE;
   "Step"[39].HMI.Display.Setpoint[0..12] := FALSE;
   "Step"[39].HMI.Display.Setpoint[13] := TRUE;
   "Step"[39].HMI.Display.Setpoint[14..15] := FALSE;
   "Step"[40].HMI.Display.Setpoint[0..15] := FALSE;
   "Step"[41].HMI.Display.Setpoint[0..15] := FALSE;
   "Step"[42].HMI.Display.Setpoint[0..15] := FALSE;
   "Step"[43].HMI.Display.Setpoint[0..15] := FALSE;
   "Step"[44].HMI.Display.Setpoint[0..15] := FALSE;
   "Step"[45].HMI.Display.Setpoint[0..15] := FALSE;
   "Step"[46].HMI.Display.Setpoint[0..15] := FALSE;
   "Step"[47].HMI.Display.Setpoint[0..15] := FALSE;
   "Step"[48].HMI.Display.Setpoint[0..15] := FALSE;
   "Step"[49].HMI.Display.Setpoint[0..15] := FALSE;
   "Step"[50].HMI.Display.Setpoint[0..15] := FALSE;
   "Step"[51].HMI.Display.Setpoint[0..15] := FALSE;
   "Step"[52].HMI.Display.Setpoint[0..15] := FALSE;
   "Step"[53].HMI.Display.Setpoint[0..15] := FALSE;
   "Step"[54].HMI.Display.Setpoint[0..15] := FALSE;
   "Step"[55].HMI.Display.Setpoint[0..15] := FALSE;
   "Step"[56].HMI.Display.Setpoint[0..15] := FALSE;
   "Step"[57].HMI.Display.Setpoint[0..15] := FALSE;
   "Step"[58].HMI.Display.Setpoint[0..15] := FALSE;
   "Step"[59].HMI.Display.Setpoint[0..15] := FALSE;
   "Step"[60].HMI.Display.Setpoint[0..15] := FALSE;
   "Step"[61].HMI.Display.Setpoint[0..15] := FALSE;
   "Step"[62].HMI.Display.Setpoint[0..12] := FALSE;
   "Step"[62].HMI.Display.Setpoint[13] := TRUE;
   "Step"[62].HMI.Display.Setpoint[14..15] := FALSE;
   "Step"[63].HMI.Display.Setpoint[0..15] := FALSE;
   "Step"[64].HMI.Display.Setpoint[0..12] := FALSE;
   "Step"[64].HMI.Display.Setpoint[13] := TRUE;
   "Step"[64].HMI.Display.Setpoint[14..15] := FALSE;
   "Step"[65].HMI.Display.Setpoint[0..15] := FALSE;
   "Step"[66].HMI.Display.Setpoint[0..12] := FALSE;
   "Step"[66].HMI.Display.Setpoint[13] := TRUE;
   "Step"[66].HMI.Display.Setpoint[14..15] := FALSE;
   "Step"[67].HMI.Display.Setpoint[0..15] := FALSE;
   "Step"[68].HMI.Display.Setpoint[0..15] := FALSE;
   Values.OperationMode := 0;
   Values.SingleStep := FALSE;
   Values.CurrentTime := 0;
   Values.CurrentStep := 0;
   Values.CycleTime := 94619;
   Values.CycleStatus := 1;
   Values.LastStep := 62;
   Values.LastVolume_1 := 15;
   Values.LastVolume_2 := 0;
   Values.IndexSelect := 10;
   Values.Vehicle[1] := '7';
   Values.Vehicle[2] := '8';
   Values.Vehicle[3..12] := '9';
   Values.Vehicle[13] := '0';
   Values.Vehicle[14] := '1';
   Values.Vehicle[15..20] := ' ';
   Values.VehicleSource := 2;
   Values.VehicleType[1] := '0';
   Values.VehicleType[2..3] := '9';
   Values.VehicleType[4..20] := ' ';
   Values.VehicleTypeSource := 5;
   Values.BufferingTime := '26.10.19  17:21:28';
   Values.DescriptionLastStep := WSTRING#'Zyklus Ende';
   Values.DescriptionActualStep := WSTRING#'Standby';
   Valve[1].Language[1..4] := WSTRING#'';
   Valve[2].Language[1..4] := WSTRING#'';
   Valve[3].Language[1..4] := WSTRING#'';
   Valve[4].Language[1..4] := WSTRING#'';
   Valve[5].Language[1..4] := WSTRING#'';
   Valve[6].Language[1..4] := WSTRING#'';
   Valve[7].Language[1..4] := WSTRING#'';
   Valve[8].Language[1..4] := WSTRING#'';
   Valve[9].Language[1..4] := WSTRING#'';
   Valve[10].Language[1] := WSTRING#'Fuellen Membranspeicher PAG Oel xxx';
   Valve[10].Language[2] := WSTRING#'charge accumulator PAG oil xxx.101';
   Valve[10].Language[3..4] := WSTRING#'';
   Valve[11].Language[1..4] := WSTRING#'';
   Valve[12].Language[1] := WSTRING#'Druckluft Pumpe R134a xxx.420';
   Valve[12].Language[2] := WSTRING#'compressed air supply (pump) R134a ';
   Valve[12].Language[3..4] := WSTRING#'';
   Valve[13].Language[1..4] := WSTRING#'';
   Valve[14].Language[1..4] := WSTRING#'';
   Valve[15].Language[1..4] := WSTRING#'';
   Valve[16].Language[1] := WSTRING#'Versorgung aus Rueckgewinnungsbehae';
   Valve[16].Language[2] := WSTRING#'Supply from recovery accumulator xx';
   Valve[16].Language[3..4] := WSTRING#'';
   Valve[17].Language[1] := WSTRING#'Rueckgewinnung Flasche xxx.384';
   Valve[17].Language[2] := WSTRING#'Recovery - Testbottle xxx.384';
   Valve[17].Language[3..4] := WSTRING#'';
   Valve[18].Language[1] := WSTRING#'Auffuellen Rueckgewinnungsbehaelter';
   Valve[18].Language[2] := WSTRING#'Charge recovery tank xxx.540';
   Valve[18].Language[3..4] := WSTRING#'';
   Valve[19].Language[1] := WSTRING#'Entleeren Abscheidebehaelter xxx.52';
   Valve[19].Language[2] := WSTRING#'discharge separator xxx.520';
   Valve[19].Language[3..4] := WSTRING#'';
   Valve[20].Language[1] := WSTRING#'Rückgewinnung / Rückgewinnung 1 - n';
   Valve[20].Language[2] := WSTRING#'Recovery - near system xxx.380';
   Valve[20].Language[3..4] := WSTRING#'';
   Valve[21].Language[1] := WSTRING#'Rückgewinnung 2 - nahe Speicher xxx';
   Valve[21].Language[2] := WSTRING#'Recovery - near tank xxx.381';
   Valve[21].Language[3..4] := WSTRING#'';
   Valve[22].Language[1..4] := WSTRING#'';
   Valve[23].Language[1] := WSTRING#'Versorgung zentral R134a xxx.20';
   Valve[23].Language[2] := WSTRING#'supply r134a xxx.20';
   Valve[23].Language[3..4] := WSTRING#'';
   Valve[24].Language[1] := WSTRING#'Versorgung zentral R134a redundant ';
   Valve[24].Language[2] := WSTRING#'supply r134a redundant xxx.21';
   Valve[24].Language[3..4] := WSTRING#'';
   Valve[25].Language[1..4] := WSTRING#'';
   Valve[26].Language[1..4] := WSTRING#'';
   Valve[27].Language[1..4] := WSTRING#'';
   Valve[28].Language[1..4] := WSTRING#'';
   Valve[29].Language[1..4] := WSTRING#'';
   Valve[30].Language[1..4] := WSTRING#'';
   Valve[31].Language[1] := WSTRING#' Fuellen vor Adapter PAG ÖL xxx.102';
   Valve[31].Language[2] := WSTRING#' Filling before adapter PAG oil xxx';
   Valve[31].Language[3..4] := WSTRING#'';
   Valve[32].Language[1..4] := WSTRING#'';
   Valve[33].Language[1..4] := WSTRING#'';
   Valve[34].Language[1..4] := WSTRING#'';
   Valve[35].Language[1..4] := WSTRING#'';
   Valve[36].Language[1..4] := WSTRING#'';
   Valve[37].Language[1..4] := WSTRING#'';
   Valve[38].Language[1..4] := WSTRING#'';
   Valve[39].Language[1..4] := WSTRING#'';
   Valve[40].Language[1..4] := WSTRING#'';
   Valve[41].Language[1..4] := WSTRING#'';
   Valve[42].Language[1..4] := WSTRING#'';
   Valve[43].Language[1] := WSTRING#'Füllen Eingang Kon R134a xxx.101';
   Valve[43].Language[2] := WSTRING#'Filling entry MU R134a xxx.101';
   Valve[43].Language[3..4] := WSTRING#'';
   Valve[44].Language[1] := WSTRING#'Fuellen vor Adapter R134a xxx.102';
   Valve[44].Language[2] := WSTRING#'filling before adapter R134a xxx.10';
   Valve[44].Language[3..4] := WSTRING#'';
   Valve[45].Language[1] := WSTRING#'Vakuumtest xxx.230';
   Valve[45].Language[2] := WSTRING#'vacuumtest xxx.230';
   Valve[45].Language[3..4] := WSTRING#'';
   Valve[46].Language[1] := WSTRING#'Vakuum xxx.200';
   Valve[46].Language[2] := WSTRING#'vacuum xxx.200';
   Valve[46].Language[3..4] := WSTRING#'';
   Valve[47].Language[1] := WSTRING#'Drucklufttest xxx.400';
   Valve[47].Language[2] := WSTRING#'compr. Air test xxx.400';
   Valve[47].Language[3..4] := WSTRING#'';
   Valve[48].Language[1..4] := WSTRING#'';
   Valve[49].Language[1] := WSTRING#'Druckluft entlasten gedrosselt xxx.';
   Valve[49].Language[2] := WSTRING#'compr. Air release throttled xxx.44';
   Valve[49].Language[3..4] := WSTRING#'';
   Valve[50].Language[1..4] := WSTRING#'';
   Valve[51].Language[1..4] := WSTRING#'';
   Valve[52].Language[1..4] := WSTRING#'';
   Valve[53].Language[1] := WSTRING#'Vakuum 1 xxx.920';
   Valve[53].Language[2] := WSTRING#'vacuum 1 xxx.920';
   Valve[53].Language[3..4] := WSTRING#'';
   Valve[54].Language[1] := WSTRING#'Fuellen 1 R134a xxx.900';
   Valve[54].Language[2] := WSTRING#'filling R134a xxx.900';
   Valve[54].Language[3..4] := WSTRING#'';
   Valve[55].Language[1] := WSTRING#'Fuellen 1 PAG xxx.900';
   Valve[55].Language[2] := WSTRING#'filling 1 PAG xxx.900';
   Valve[55].Language[3..4] := WSTRING#'';
   Valve[56].Language[1] := WSTRING#'Stoeßel 1 xxx.960';
   Valve[56].Language[2] := WSTRING#'plunger 1 xxx.960';
   Valve[56].Language[3..4] := WSTRING#'';
   Valve[57].Language[1] := WSTRING#'Verriegeln 1 xxx.940';
   Valve[57].Language[2] := WSTRING#'clamping 1 xxx.940';
   Valve[57].Language[3..4] := WSTRING#'';
   Valve[58].Language[1..4] := WSTRING#'';
   Valve[59].Language[1..4] := WSTRING#'';
   Valve[60].Language[1] := WSTRING#'Vakuum 2 xxx.1010';
   Valve[60].Language[2] := WSTRING#'vacuum 2 xxx.1010';
   Valve[60].Language[3..4] := WSTRING#'';
   Valve[61].Language[1] := WSTRING#'Stoeßel 2 xxx.1040';
   Valve[61].Language[2] := WSTRING#'plunger 2 xxx.1040';
   Valve[61].Language[3..4] := WSTRING#'';
   Valve[62].Language[1] := WSTRING#'Verriegeln 2 xxx.1020';
   Valve[62].Language[2] := WSTRING#'clamping 2 xxx.1020';
   Valve[62].Language[3..4] := WSTRING#'';
   Valve[63].Language[1..4] := WSTRING#'';
   Valve[64].Language[1..4] := WSTRING#'';
   Valve[1..9].Status := FALSE;
   Valve[10].Status := TRUE;
   Valve[11].Status := FALSE;
   Valve[12].Status := TRUE;
   Valve[13..15].Status := FALSE;
   Valve[16..21].Status := TRUE;
   Valve[22].Status := FALSE;
   Valve[23..24].Status := TRUE;
   Valve[25..30].Status := FALSE;
   Valve[31].Status := TRUE;
   Valve[32..42].Status := FALSE;
   Valve[43..47].Status := TRUE;
   Valve[48].Status := FALSE;
   Valve[49].Status := TRUE;
   Valve[50..52].Status := FALSE;
   Valve[53..57].Status := TRUE;
   Valve[58..59].Status := FALSE;
   Valve[60..62].Status := TRUE;
   Valve[63..64].Status := FALSE;
   ParaInfo[1].ParaName[1] := WSTRING#'Vakuum [mbar]';
   ParaInfo[1].ParaName[2] := WSTRING#'vacuum [mbar]';
   ParaInfo[1].ParaName[3..4] := WSTRING#'';
   ParaInfo[2].ParaName[1] := WSTRING#'Delta Vakuum [mbar]';
   ParaInfo[2].ParaName[2] := WSTRING#'delta vacuum [mbar]';
   ParaInfo[2].ParaName[3..4] := WSTRING#'';
   ParaInfo[3].ParaName[1..4] := WSTRING#'';
   ParaInfo[4].ParaName[1..4] := WSTRING#'';
   ParaInfo[5].ParaName[1] := WSTRING#'Test Druck [mbar]';
   ParaInfo[5].ParaName[2] := WSTRING#'test pressure [mbar]';
   ParaInfo[5].ParaName[3..4] := WSTRING#'';
   ParaInfo[6].ParaName[1] := WSTRING#'Delta Test Druck [mbar]';
   ParaInfo[6].ParaName[2] := WSTRING#'Delta test pressure [mbar]';
   ParaInfo[6].ParaName[3..4] := WSTRING#'';
   ParaInfo[7].ParaName[1] := WSTRING#'Masse R134a [g]';
   ParaInfo[7].ParaName[2] := WSTRING#'mass R134a [g]';
   ParaInfo[7].ParaName[3..4] := WSTRING#'';
   ParaInfo[8].ParaName[1] := WSTRING#'Menge PAG [ml]';
   ParaInfo[8].ParaName[2] := WSTRING#'volume PAG [ml]';
   ParaInfo[8].ParaName[3..4] := WSTRING#'';
   ParaInfo[9].ParaName[1..4] := WSTRING#'';
   ParaInfo[10].ParaName[1..4] := WSTRING#'';
   ParaInfo[11].ParaName[1..4] := WSTRING#'';
   ParaInfo[12].ParaName[1..4] := WSTRING#'';
   ParaInfo[13].ParaName[1] := WSTRING#'Proportionalventil Druckluft [mbar]';
   ParaInfo[13].ParaName[2] := WSTRING#'proportional valve compr. air [mbar';
   ParaInfo[13].ParaName[3..4] := WSTRING#'';
   ParaInfo[14].ParaName[1..4] := WSTRING#'';
   ParaInfo[15].ParaName[1..4] := WSTRING#'';
   ParaInfo[1..2].Factor := 10;
   ParaInfo[3..15].Factor := 1;
   ParaInfo[1..2].DecimalPoint := 1;
   ParaInfo[3..15].DecimalPoint := 0;
END_DATA_BLOCK
